TYPE PM101OpticalPowermeterConfig EXTENDS DeviceConfiguration :
STRUCT
	SerialCommunication : SerialCommunication;
	Sensor : PowermeterSensor;
END_STRUCT
END_TYPE

(* stored: Version 1.1.0.1, ProductVersion 3.1.4024.10
   DUT PM101OpticalPowermeterConfig: Id {d09785e0-a5fa-4a72-be45-a87bdc433a8f} *)
